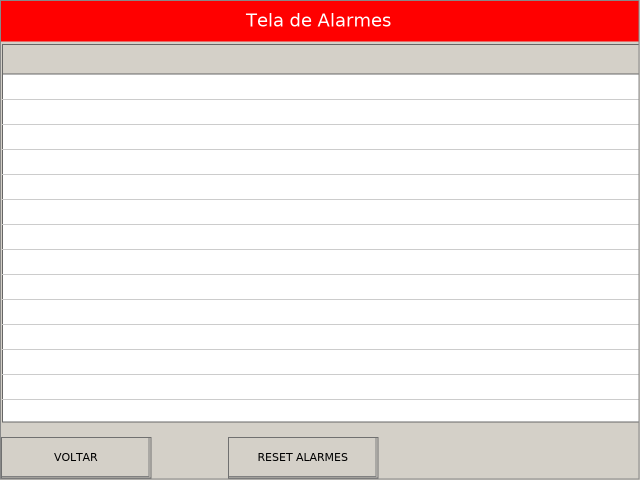
VISUALIZATION VISU_ALARMS  // 640x480
    Button (1,437 150x41), "VOLTAR"
        OnMouseClick: change screen: VISU_MAIN
    Rectangle (-1,0 640x41), "Tela de Alarmes"
    Button (228,437 150x41), "RESET ALARMES"
        tap GVL_ALARMS.bResetAlarms
    Table (2,44 637x378), data array: GVL_ALARMS.ACTIVE_ALARMS
        p746581629: GVL_ALARMS.HISTORY_ALARMS[INDEX].dwTextColor
        p3854506369: GVL_ALARMS.ACTIVE_ALARMS[INDEX].byAckStatus
        p1892666644: GVL_ALARMS.ACTIVE_ALARMS[INDEX].byGroup
        p338671338: ACTIVE_ALARMS[INDEX].sDate
        p2170511999: GVL_ALARMS.ACTIVE_ALARMS[INDEX].sHour
        p3723444502: GVL_ALARMS.ACTIVE_ALARMS[INDEX].iNumber
        p1218418051: GVL_ALARMS.ACTIVE_ALARMS[INDEX].dwTextColor
        p2232123230: !
        p1791247317: GVL_ALARMS.ACTIVE_ALARMS[INDEX].sDate
END_VISUALIZATION

(* stored: Version 1.1.0.1, ProductVersion 3.1.4024.12
   Visu VISU_ALARMS: Id {4b1d3678-66c5-4c86-b2bf-d3e64f0331ee} *)
